% RSLogix 500 project PLC_1_LAB6-1.RSS, saved by version 12.00.00.00 %
PROJECT "UNTITLED"    % processor: Bul.1763 MicroLogix 1100 Series B %

PROGRAM FILES
  LAD 2   11 rungs

DATA FILES
  O0 OUTPUT  5 elements
  I1 INPUT  6 elements
  S2 STATUS  66 elements
  B3 BINARY  1 elements
  T4 TIMER  3 elements
  C5 COUNTER  3 elements
  R6 CONTROL  1 elements
  N7 INTEGER  1 elements
  F8 FLOAT  1 elements

LADDER 2
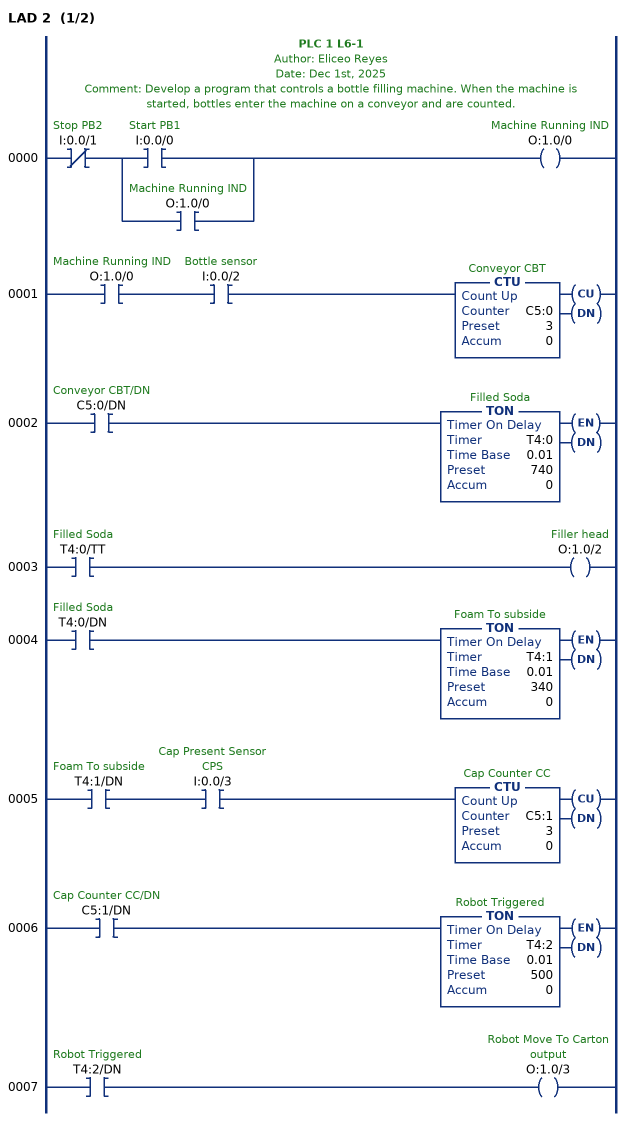
% Rung: 0 %
% TITLE: PLC 1 L6-1 %
% Author: Eliceo Reyes
% Date: Dec 1st, 2025
% Comment: Develop a program that controls a bottle filling machine. When the machine is started, bottles enter the machine on a conveyor and are counted. %
SOR XIO I:0.0/1 BST XIC I:0.0/0 NXB XIC O:1.0/0 BND OTE O:1.0/0 EOR
%   I:0.0/1  PB2  "Stop" %
%   I:0.0/0  PB1  "Start" %
%   O:1.0/0  IND  "Machine Running" %
% Rung: 1 %
SOR XIC O:1.0/0 XIC I:0.0/2 CTU C5:0 3 0 EOR
%   O:1.0/0  IND  "Machine Running" %
%   I:0.0/2  "Bottle sensor" %
%   C5:0  CBT  "Conveyor" %
% Rung: 2 %
SOR XIC C5:0/DN TON T4:0 0.01 740 0 EOR
%   C5:0  CBT  "Conveyor" %
%   T4:0  "Filled Soda" %
% Rung: 3 %
SOR XIC T4:0/TT OTE O:1.0/2 EOR
%   T4:0  "Filled Soda" %
%   O:1.0/2  "Filler head" %
% Rung: 4 %
SOR XIC T4:0/DN TON T4:1 0.01 340 0 EOR
%   T4:0  "Filled Soda" %
%   T4:1  "Foam To subside" %
% Rung: 5 %
SOR XIC T4:1/DN XIC I:0.0/3 CTU C5:1 3 0 EOR
%   T4:1  "Foam To subside" %
%   I:0.0/3  CPS  "Cap Present Sensor" %
%   C5:1  CC  "Cap Counter" %
% Rung: 6 %
SOR XIC C5:1/DN TON T4:2 0.01 500 0 EOR
%   C5:1  CC  "Cap Counter" %
%   T4:2  "Robot Triggered" %
% Rung: 7 %
SOR XIC T4:2/DN OTE O:1.0/3 EOR
%   T4:2  "Robot Triggered" %
%   O:1.0/3  "Robot Move To Carton output" %

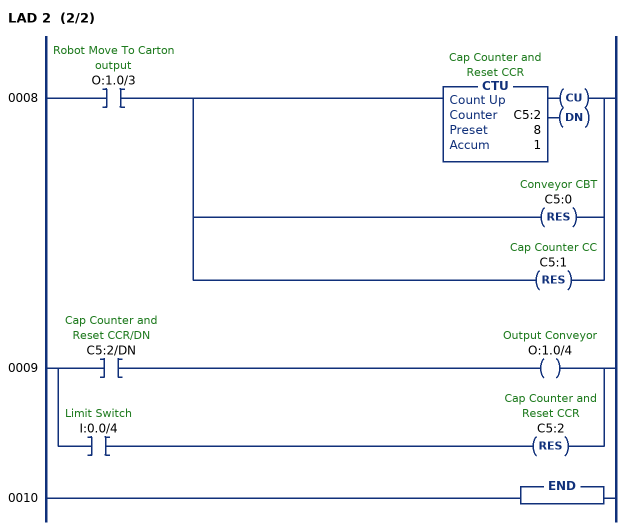
% Rung: 8 %
SOR XIC O:1.0/3 BST CTU C5:2 8 1 NXB RES C5:0 NXB RES C5:1 BND EOR
%   O:1.0/3  "Robot Move To Carton output" %
%   C5:2  CCR  "Cap Counter and Reset" %
%   C5:0  CBT  "Conveyor" %
%   C5:1  CC  "Cap Counter" %
% Rung: 9 %
SOR BST XIC C5:2/DN OTE O:1.0/4 NXB XIC I:0.0/4 RES C5:2 BND EOR
%   C5:2  CCR  "Cap Counter and Reset" %
%   O:1.0/4  "Output Conveyor" %
%   I:0.0/4  "Limit Switch" %
% Rung: 10 %
SOR END EOR

OTHER DOCUMENTED ADDRESSES
  XIC  
  XIO  

DATA TABLE (non-zero values as saved)
DATA T4
% .PRE .ACC %
% T4:0 % 740 0
% T4:1 % 340 0
% T4:2 % 500 0
DATA C5
% .PRE .ACC %
% C5:0 % 3 0
% C5:1 % 3 0
% C5:2 % 8 1
